Staubli VAL3: atiForceSen7.dtx

bool bClear
bool bOverRun
public bool bZero
mdesc mNomSpeed
public num nForce[6]
num nHeader[2]
num nMonitor[2]
num nPort = 49151
num nRec[16]
num nReceived = -1
num nScaleForce = 6104
num nScaleTorque = 153
num nSend[20]
num nSent = -1
num nSioTimeOut = 5
public num nStatus
num nVecForce
sio sFs = {link=Socket\sAtiFs}
num nCountPerFs
num nCountPerTq
